Yaskawa INFORM job: X2_25(90,90).JBI

/JOB
//NAME X2_25(90,90)
//POS
///NPOS 42,42,42,3,0,0
///TOOL 0
///POSTYPE PULSE
///PULSE
C00000=-2027,-78555,-65913,-1,89981,-9
C00001=38531,-95764,-73065,32205,93197,-48118
C00002=43402,-96116,-70716,32673,89950,-47114
C00003=45387,-95531,-68532,32857,88301,-46804
C00004=45383,-95077,-67593,32856,88011,-46890
C00005=45387,-95269,-67962,32857,88118,-46857
C00006=46822,-97938,-68938,32997,86912,-46639
C00007=45387,-95269,-67962,32857,88118,-46857
C00008=36831,-101714,-70295,31838,89769,-49757
C00009=37431,-98465,-67310,31918,89401,-49626
C00010=38568,-97705,-67036,32074,89165,-49247
C00011=36268,-99209,-67576,31752,89648,-50011
C00012=29459,-100543,-74819,30874,95404,-51093
C00013=20675,-116676,-87310,22832,76539,-34670
C00014=42270,-104866,-76555,9210,50261,-7718
C00015=43428,-96605,-71126,8511,51029,-7146
C00016=43846,-92977,-67993,8306,50922,-6974
C00017=43842,-92440,-66827,8360,50486,-7013
C00018=43809,-92717,-67354,8355,50669,-7011
C00019=42526,-89985,-66292,8913,51548,-7489
C00020=43809,-92717,-67354,8355,50669,-7011
C00021=35228,-99076,-69732,12914,50018,-10840
C00022=36629,-97765,-66398,12477,48455,-10422
C00023=37968,-96893,-66082,11755,48504,-9814
C00024=35668,-98364,-66614,12992,48433,-10859
C00025=35228,-99076,-69732,12914,50018,-10840
C00026=57676,-71636,-58241,-5950,65068,10540
C00027=64200,-66759,-55921,-12568,68748,18582
C00028=63297,-67618,-56325,-11636,68043,17382
C00029=65085,-65455,-55213,-13109,69308,19287
C00030=67037,-63366,-54254,-15446,71445,22505
C00031=67026,-63387,-54264,-15444,71439,22502
C00032=37931,-107129,-85744,4222,83758,-27344
C00033=66770,-63887,-54522,21209,99670,-56787
C00034=66768,-63894,-54526,21209,99670,-56788
C00035=66213,-64902,-54857,21108,99519,-57020
C00036=65282,-66699,-55945,20957,99519,-57364
C00037=66767,-63896,-54527,21209,99669,-56788
C00038=67429,-62591,-53856,21318,99737,-56530
C00039=66768,-63894,-54525,21209,99670,-56788
C00040=66771,-63887,-54522,21209,99670,-56787
C00041=-2027,-78555,-65913,-1,89981,-9
BC00000=1577,523905,619430
BC00001=25181,438263,219567
BC00002=25181,438263,219567
BC00003=25181,438263,219567
BC00004=25181,438263,219567
BC00005=25181,438263,219567
BC00006=25181,438263,219567
BC00007=25181,438263,219567
BC00008=25181,438263,219567
BC00009=25181,438263,219567
BC00010=25181,438263,219567
BC00011=25181,438263,219567
BC00012=25181,438263,219567
BC00013=133625,437775,218883
BC00014=244352,437277,218186
BC00015=244352,437277,218186
BC00016=244352,437277,218186
BC00017=244352,437277,218186
BC00018=244352,437277,218186
BC00019=244352,437277,218186
BC00020=244352,437277,218186
BC00021=244352,437277,218186
BC00022=244352,437277,218186
BC00023=244352,437277,218186
BC00024=244352,437277,218186
BC00025=244352,437277,218186
BC00026=246001,450309,249218
BC00027=246016,445701,249197
BC00028=246022,443704,249188
BC00029=246037,439095,249166
BC00030=243792,439354,256742
BC00031=238180,439999,275681
BC00032=134467,443567,275053
BC00033=30898,451321,275535
BC00034=25291,450641,256593
BC00035=23048,450370,249016
BC00036=23063,445762,248995
BC00037=23067,444364,248988
BC00038=23082,439755,248967
BC00039=25325,440027,256543
BC00040=30933,440706,275485
BC00041=1577,523905,619430
EC00000=-798156,-740307
EC00001=-798156,-740307
EC00002=-798156,-740307
EC00003=-798156,-740307
EC00004=-798156,-740307
EC00005=-798156,-740307
EC00006=-798156,-740307
EC00007=-798156,-740307
EC00008=-798156,-740307
EC00009=-798156,-740307
EC00010=-798156,-740307
EC00011=-798156,-740307
EC00012=-798156,-740307
EC00013=-798156,-740307
EC00014=-798156,-740307
EC00015=-798156,-740307
EC00016=-798156,-740307
EC00017=-798156,-740307
EC00018=-798156,-740307
EC00019=-798156,-740307
EC00020=-798156,-740307
EC00021=-798156,-740307
EC00022=-798156,-740307
EC00023=-798156,-740307
EC00024=-798156,-740307
EC00025=-798156,-740307
EC00026=-798156,-740307
EC00027=-798156,-740307
EC00028=-798156,-740307
EC00029=-798156,-740307
EC00030=-798156,-740307
EC00031=-798156,-740307
EC00032=-798156,-740307
EC00033=-798156,-740307
EC00034=-798156,-740307
EC00035=-798156,-740307
EC00036=-798156,-740307
EC00037=-798156,-740307
EC00038=-798156,-740307
EC00039=-798156,-740307
EC00040=-798156,-740307
EC00041=-798156,-740307
///POSTYPE BASE
///RECTAN
///RCONF 0,0,0,0,1,0,0,0,0,0,0,0,0,0,0,0,0,0,0,0,0,0,0,0
P00006=2.006,1.622,-0.565,0.0000,0.0000,0.0000
P00021=0.073,2.058,-0.109,0.0000,0.0000,0.0000
P00022=2.006,1.622,-0.565,0.0000,0.0000,0.0000
//INST
///DATE 2024/12/16 22:01
///ATTR SC,RW
///GROUP1 RB1,BS1
///GROUP2 ST1
NOP
'X2_25(90,90)
MOVJ C00000 BC00000 VJ=100.00  +MOVJ EC00000 VJ=100.00
'Path S3561
SFTOF3D
MOVJ C00001 BC00001 VJ=100.00  +MOVJ EC00001 VJ=100.00
MOVL C00002 BC00002 V=800.0  +MOVJ EC00002 VJ=100.00
SMOVL C00003 BC00003 V=166.7  +MOVJ EC00003
SREFP 3 C00004 BC00004  +REFP EC00004
CALL JOB:SEARCH-R1-S13D
SET P022 P006
SFTON3D P022
SMOVL C00005 BC00005 V=166.7  +MOVJ EC00005
SREFP 3 C00006 BC00006  +REFP EC00006
CALL JOB:SEARCH-R1-S13D
SET P022 P006
SFTON3D P022
SMOVL C00007 BC00007 V=166.7  +MOVJ EC00007
SMOVL C00008 BC00008 V=166.7  +MOVJ EC00008
SMOVL C00009 BC00009 V=166.7  +MOVJ EC00009
SREFP 3 C00010 BC00010  +REFP EC00010
CALL JOB:SEARCH-R1-S13D
SET P022 P006
SFTON3D P022
SMOVL C00011 BC00011 V=166.7  +MOVJ EC00011
MOVL C00012 BC00012 V=1000.0  +MOVJ EC00012 VJ=100.00
'EndPath S3561
MOVJ C00013 BC00013 VJ=100.00  +MOVJ EC00013 VJ=100.00
'Path S3562
SFTOF3D
MOVJ C00014 BC00014 VJ=100.00  +MOVJ EC00014 VJ=100.00
MOVL C00015 BC00015 V=800.0  +MOVJ EC00015 VJ=100.00
SMOVL C00016 BC00016 V=166.7  +MOVJ EC00016
SREFP 3 C00017 BC00017  +REFP EC00017
CALL JOB:SEARCH-R1-S13D
SET P021 P006
SFTON3D P021
SMOVL C00018 BC00018 V=166.7  +MOVJ EC00018
SREFP 3 C00019 BC00019  +REFP EC00019
CALL JOB:SEARCH-R1-S13D
SET P021 P006
SFTON3D P021
SMOVL C00020 BC00020 V=166.7  +MOVJ EC00020
SMOVL C00021 BC00021 V=250.0  +MOVJ EC00021
SMOVL C00022 BC00022 V=166.7  +MOVJ EC00022
SREFP 3 C00023 BC00023  +REFP EC00023
CALL JOB:SEARCH-R1-S13D
SET P021 P006
SFTON3D P021
SMOVL C00024 BC00024 V=166.7  +MOVJ EC00024
SMOVL C00025 BC00025 V=500.0  +MOVJ EC00025
'EndPath S3562
'Path W3563
SFTOF3D
SFTON3D P021
SMOVL C00026 BC00026 V=166.7 PL=0  +MOVJ EC00026
MACRO1 MJ#(0) ARGF9
ARCON
SMOVL C00027 BC00027 V=8.3  +MOVJ EC00027
SMOVL C00028 BC00028 V=8.3  +MOVJ EC00028
SMOVL C00029 BC00029 V=8.3  +MOVJ EC00029
ARCOF
SMOVL C00030 BC00030 V=800.0  +MOVJ EC00030
SMOVL C00031 BC00031 V=1000.0  +MOVJ EC00031
SFTOF3D
'EndPath W3563
MOVJ C00032 BC00032 VJ=100.00  +MOVJ EC00032 VJ=100.00
'Path W3564
SFTOF3D
SFTON3D P022
MOVJ C00033 BC00033 VJ=100.00  +MOVJ EC00033 VJ=100.00
SMOVL C00034 BC00034 V=800.0  +MOVJ EC00034
SMOVL C00035 BC00035 V=166.7 PL=0  +MOVJ EC00035
ARCON
SMOVL C00036 BC00036 V=9.2  +MOVJ EC00036
SMOVL C00037 BC00037 V=9.2  +MOVJ EC00037
SMOVL C00038 BC00038 V=9.2  +MOVJ EC00038
ARCOF
SMOVL C00039 BC00039 V=800.0  +MOVJ EC00039
SMOVL C00040 BC00040 V=1000.0  +MOVJ EC00040
SFTOF3D
'EndPath W3564
MOVJ C00041 BC00041 VJ=100.00  +MOVJ EC00041 VJ=100.00
END
